Staubli VAL3: remGetIPVals.pgx

program remGetIPVals(string& sReturn[] (dimensions=1))
  local trsf trIP
begin
  // Return the values of the active interaction point.
  //
  logMsg("call remGetIPVals")
  if nIPNumber==0
    trIP=fIP1.trsf
  else
    trIP=fIP2.trsf
  endIf
  sReturn="GETIPVALS"
  sReturn=sReturn+" "+toString(sNumConv,trIP.x)
  sReturn=sReturn+" "+toString(sNumConv,trIP.y)
  sReturn=sReturn+" "+toString(sNumConv,trIP.z)
  sReturn=sReturn+" "+toString(sNumConv,trIP.rx)
  sReturn=sReturn+" "+toString(sNumConv,trIP.ry)
  sReturn=sReturn+" "+toString(sNumConv,trIP.rz)
end
